INTERFACE I_CtrlBase

METHOD iniCtrlArray : BOOL
VAR_INPUT
	p_pCtrlArray: POINTER TO POINTER TO fb_CtrlBase;
	intCtrlID: INT;
END_VAR
END_METHOD

METHOD getCtrlCIf : POINTER TO T_Ctrl_CIf
END_METHOD

END_INTERFACE

(* stored: Version 1.1.0.1, ProductVersion 3.1.0.18
   Itf I_CtrlBase: Id {f33ff886-408d-4d15-bdc3-596cc3f70de4}
   Method iniCtrlArray: Id {4446fe44-dee4-4d83-99ed-7d6d0073c8b5}
   Method getCtrlCIf: Id {daad236f-6b83-4f69-bc88-4edd98c0c85a} *)
